FUNCTION_BLOCK FB_Outer EXTENDS FB_Parameters_Base
VAR
	middler	: FB_Middler(THIS^);
END_VAR

END_FUNCTION_BLOCK

(* stored: Version 1.1.0.1, ProductVersion 3.1.4024.15
   POU FB_Outer: Id {5e67aabd-87b3-4e95-a45a-fe2aebd34d5d}, SpecialFunc None *)
